// TIA Portal V19 export
DATA_BLOCK "PUMP SELECTION"   // DB19
{ S7_Optimized_Access := 'FALSE' }
   VAR RETAIN
      "MGF FEED PUMP P-101 A/B" : Bool;
      "MGF FEED PUMP P-102 A/B" : Bool;
      "UF FEED PUMP P-103 A/B" : Bool;
      "UF BLOWER AB-201 A/B" : Bool;
      "UF BACK WASH P-201 A/B" : Bool;
      "DM FEED PUMP P-502 A" : Bool;
      "DM FEED PUMP P-502 B" : Bool;
      "DM FEED PUMP P-502 C" : Bool;
      "BACK WASH RECOVERY P-801 A/B" : Bool;
      "NaOCL DOSING D-706 A/B" : Bool;
   END_VAR
BEGIN
END_DATA_BLOCK
